Fanuc TP program (LS listing): RESET_PR.LS

/PROG  RESET_PR
/ATTR
OWNER		= MNEDITOR;
COMMENT		= "(PR)";
PROG_SIZE	= 202;
CREATE		= DATE 22-11-17  TIME 19:36:22;
MODIFIED	= DATE 22-12-14  TIME 22:20:34;
FILE_NAME	= ;
VERSION		= 0;
LINE_COUNT	= 4;
MEMORY_SIZE	= 558;
PROTECT		= READ_WRITE;
TCD:  STACK_SIZE	= 0,
      TASK_PRIORITY	= 50,
      TIME_SLICE	= 0,
      BUSY_LAMP_OFF	= 0,
      ABORT_REQUEST	= 0,
      PAUSE_REQUEST	= 0;
DEFAULT_GROUP	= 1,*,*,*,*;
CONTROL_CODE	= 00000000 00000000;
/MN
   1:  FOR R[200:#]=1 TO 6 ;
   2:  PR[AR[1],R[200]]=0    ;
   3:  ENDFOR ;
   4:  R[200:#]=0    ;
/POS
/END
